FUNCTION_BLOCK Q_BackgroundColour (* Command change background colour ( Part 6 - F.20 ) *)
  (* Standard: ISO 11783-6; Description: Copyright (c) 2022 HR Agrartechnik GmbH This program and the accompanying materials are made available under the terms of the Eclipse Public License 2.0 which is available at https://www.eclipse.org/legal/epl-2.0/ SPDX-License-Identifier: EPL-2.0 see Description Tab *)
  (* Version 1.0, 2022-07-08, Franz Höpfinger, HR Agrartechnik GmbH *)
  PACKAGE isobus::UT::Q;
  IMPORT isobus::UT::Q::const::IDs::ID_NULL;
  (* Documentation:
  Command change background colour ( Part 6 - F.20 )
   This command is used to change the background colour of an object.
   Valid Object IDs
   A background colour Object ID is valid if it falls within one of the following ISO 11783-6 ID ranges:
    - WorkingSet: 0
   - DataMask: 1000 – 1999
   - AlarmMask: 2000 – 2999
   - SoftKeyMask: 4000 – 4999
   - Key: 5000 – 5999
   - Button: 6000 – 6999
   - InputBooleanField: 7000 – 7999
   - InputStringField: 8000 – 8999
   - InputNumberField: 9000 – 9999
   - OutputStringField: 11000 – 11999
   - OutputNumberField: 12000 – 12999
   - WindowMaskObject: 34000 – 34999
   - GraphicsContextObject: 36000 – 36999
   - AuxiliaryFunction: 29000 – 29999
   - AuxiliaryFunctionType2: 31000 – 31999
   - AuxiliaryInputType2: 32000 – 32999
    ID_NULL (65535) is not a command target but can be used in INIT to deactivate the FB. Any ID outside these ranges is invalid for commanding.
   Activate / Deactivate
   The FB is deactivated by default. It becomes active when INIT provides a valid background colour Object ID. Sending INIT with ID_NULL (65535) deactivates the FB again. This toggle can be repeated arbitrarily.
    - INIT + ID_NULL (65535): FB deactivated, STATUS="DEACTIVATED", s16result=VT_E_DEACTIVATED (-40)
   - INIT + valid background colour ID: FB activated, STATUS="initialized", s16result=VT_E_NO_ERR (0). If a REQ was buffered before, it is executed immediately.
   - INIT + invalid ID: STATUS="ERROR: Invalid Object ID (not a background colour object)", s16result=VT_E_INVALID_OBJECT_ID (-132)
    REQ Handling
    - REQ before any INIT: Buffered, STATUS="Buffered: INIT not yet completed", s16result=VT_E_NOT_READY (-131)
   - REQ while deactivated (INIT came with NULL or invalid ID): STATUS shows the actual deactivation reason, s16result=VT_E_DEACTIVATED (-40) or VT_E_INVALID_OBJECT_ID (-132)
   - REQ while active: Command sent to VT, result reflected in CNF
    param[in] {u16ObjId, uint16_t}
   Object ID. Use ID_NULL (65535) to deactivate the FB. Use a valid background colour object ID to activate.
   param[in] {u8Colour, uint8_t}
   New Background colour see Part 6 - A.3 VT standard colour palette
   Return Values (s16result):
   int16_t
    - VT_E_NO_ERR (0) - OK
   - VT_E_DEACTIVATED (-40) - FB deactivated (INIT received with ID_NULL)
   - VT_E_INVALID_OBJECT_ID (-132) - Object ID is invalid (not a background colour object)
   - VT_E_NOT_READY (-131) - Buffered: INIT not yet completed
   - VT_E_OVERFLOW (-6) - buffer overflow
   - VT_E_NOACT (-8) - Command not possible in current state
   - VT_E_NO_INSTANCE (-21) - No VT client available
   - VT_E_ISO_INSTANCE_INVALID (-129) - Identifier for instance (connection) invalid
   - VT_E_HANDLE_INVALID (-128) - ErrorCause: invalid Handle
   - VT_E_NOT_ALIVE (-130) - Identifier for instance valid, but VT Dead.
    Instanz-Eindeutigkeit (Instance Uniqueness)
   Dieser Baustein erfordert Instanz-Eindeutigkeit bezüglich u16ObjId. Es darf im gesamten Programm nur eine Instanz von Q_BackgroundColour für dieselbe Ziel-Objekt-ID existieren (kann dieselbe ID mit EINER Q_BackgroundColourAux-Instanz teilen, da unterschiedliche FB-Klassen, aber niemals zwei Q_BackgroundColour-Instanzen auf dieselbe ID).
  *)
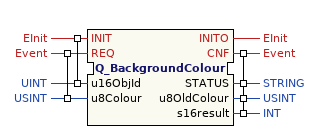
  EVENT_INPUT
    INIT : EInit WITH u16ObjId; (* Service Initialization *)
    REQ WITH u8Colour; (* Service Request *)
  END_EVENT
  EVENT_OUTPUT
    INITO : EInit; (* Initialization Confirm *)
    CNF WITH STATUS, u8OldColour, s16result; (* Confirmation of Requested Service *)
  END_EVENT
  VAR_INPUT
    u16ObjId : UINT := ID_NULL; (* Object ID *)
    u8Colour : USINT; (* New Background colour see Part 6 - A.3 VT standard colour palette *)
  END_VAR
  VAR_OUTPUT
    STATUS : STRING; (* Service Status *)
    u8OldColour : USINT; (* Old value of ID *)
    s16result : INT; (* retval see description *)
  END_VAR
END_FUNCTION_BLOCK
